{attribute 'qualified_only'}
{attribute 'strict'}
TYPE DUT :
(
	enum_member := 0
);
END_TYPE

(* stored: Version 1.1.0.1, ProductVersion 3.1.4024.12
   DUT DUT: Id {e7f2fda9-fae7-4f52-bf65-ca37665b8314} *)
